Fanuc KAREL source: kt00447.KL

-- PROVISIONAL review KL for V770-1; original PC SHA256 41c9cdce1a8877edf472cee20595339c89b6349abf53e685cd10497b479cb5f6
-- Incomplete behavior may be omitted. Consult companion uncertainty JSON. Do not deploy.
PROGRAM KT00447
%NOLOCKGROUP
VAR
  I2 : INTEGER
  OUT : BOOLEAN
-- UNRESOLVED_DECL Y1 type=002018
BEGIN
  -- UNRESOLVED_PC offsets 5-19; opcodes 2E,22,9D,33,B2
  -- UNRESOLVED_PC offsets 24-35; opcodes 2E,23
  -- UNRESOLVED_PC offsets 40-62; opcodes 22,9D,33,B1,21,5C,23
  -- UNRESOLVED_PC offsets 67-71; opcodes 7F
END KT00447
